FUNCTION_BLOCK FB_PowerNC_TestDouble IMPLEMENTS  I_Power
VAR
    bError : BOOL;
    nErrorID : UDINT := 18000;
END_VAR

PROPERTY Aborted : BOOL
GET
END_GET
END_PROPERTY

PROPERTY Active : BOOL
GET
END_GET
END_PROPERTY

PROPERTY Busy : BOOL
GET
END_GET
END_PROPERTY

METHOD DisablePower
END_METHOD

PROPERTY Done : BOOL
GET
END_GET
END_PROPERTY

PROPERTY Error : BOOL
GET
Error := bError;
END_GET
SET
bError := Error;
END_SET
END_PROPERTY

PROPERTY ErrorID : UDINT
GET
ErrorId := nErrorID;
END_GET
SET
nErrorId := ErrorID;
END_SET
END_PROPERTY

PROPERTY Message : T_MAXSTRING
GET
END_GET
END_PROPERTY

PROPERTY Override : LREAL
GET
END_GET
END_PROPERTY

METHOD Power
VAR_INPUT
    Enable	: BOOL;
    Enable_Positive	: BOOL;
    Enable_Negative	: BOOL;
    Override	: LREAL := 100;
    BufferMode	: MC_BufferMode := .MC_BufferMode.MC_Aborting;
END_VAR
END_METHOD

PROPERTY PowerIsEnabled : BOOL
GET
PowerIsEnabled := TRUE;
END_GET
END_PROPERTY

END_FUNCTION_BLOCK

(* stored: Version 1.1.0.1
   POU FB_PowerNC_TestDouble: Id {e2657803-eb37-4d34-9ec3-385056392f02}, SpecialFunc None
   Property Aborted: Id {588c075c-cd02-4a46-a82a-f9a27dd32a85}
   Get Get: Id {b2824654-2943-419b-a4b9-5391622b456e}
   Property Active: Id {4a4271ec-3e2a-4139-b786-f1aa6837aee6}
   Get Get: Id {2062f7aa-dd6e-4089-aeed-074ac4ccdd17}
   Property Busy: Id {3ac7eba8-0cd3-472c-91dc-f2d9e7a9703f}
   Get Get: Id {b325d860-039c-4ba2-bb69-23b2aa11fecf}
   Method DisablePower: Id {a3f7a0f3-1c59-4d6c-9253-c0a1c22e7ba1}
   Property Done: Id {e7e0839c-647c-4e91-bdff-feff9fbf51ae}
   Get Get: Id {d7c51040-3c34-431a-8805-c3582ce9ebb0}
   Property Error: Id {4ecab9c3-1d3d-47e7-9717-e97ecd103123}
   Get Get: Id {18f168e9-b54c-4e16-bfd0-429ca7b54f9c}
   Set Set: Id {754c2e90-8695-4d77-b05f-6e6bf1eac737}
   Property ErrorID: Id {8b324087-df58-4aa3-b156-fc71a4873f92}
   Get Get: Id {9805a0a1-324c-44df-a348-5c6f21faca9e}
   Set Set: Id {dbd077b5-d855-4b2a-b77c-63d36dfa09a7}
   Property Message: Id {62099cf1-cd9c-4bf1-aee6-a9cbd9250d3b}
   Get Get: Id {e97b9d4b-1df1-4f85-b010-5a5f401a0a79}
   Property Override: Id {31807e1c-756f-4cde-a51b-fd20b717c119}
   Get Get: Id {2db10e6f-30f0-4665-8905-e7250e73d402}
   Method Power: Id {19e3e1be-8ca4-4b90-a1b4-d997fa9320db}
   Property PowerIsEnabled: Id {9f031727-b2fa-4bfb-b74b-1d9537057a10}
   Get Get: Id {b3c7f030-178b-40a2-ae22-c9a17b0b1823} *)
